// TIA Portal V15.1 export
// export: Created 2020-12-23T11:47:33.918068Z, ExportSetting WithDefaults, WithReadOnly, DisplayName Totally Integrated Automation Portal, DisplayVersion V15.1 Update 3, DisplayName TIA Portal Openness, DisplayVersion V15.1, DisplayName STEP 7 Professional, DisplayVersion V15.1 Update 3, DisplayName WinCC Advanced, DisplayVersion V15.1 Update 3
VAR_GLOBAL   // PLC tag table "io_import"
   "VSEN TBL TABLE LH HP UP" AT I60.0 : Bool;   // #nc - VSEN TBL TABLE LH HP UP
   "VSEN TBL TABLE LH WP DOWN" AT I61.0 : Bool;   // #nc - VSEN TBL TABLE LH WP DOWN
   "VALVE TBL TABLE LH HP UP" AT Q60.6 : Bool;   // [1] VALVE TBL TABLE LH HP UP
   "VALVE TBL TABLE LH WP DOWN" AT Q61.6 : Bool;   // [1] VALVE TBL TABLE LH WP DOWN
   "VSEN TBL TABLE RH HP UP" AT I60.1 : Bool;   // #nc - VSEN TBL TABLE RH HP UP
   "VSEN TBL TABLE RH WP DOWN" AT I61.1 : Bool;   // #nc - VSEN TBL TABLE RH WP DOWN
   "VALVE TBL TABLE RH HP UP" AT Q60.7 : Bool;   // [2] VALVE TBL TABLE RH HP UP
   "VALVE TBL TABLE RH WP DOWN" AT Q61.7 : Bool;   // [2] VALVE TBL TABLE RH WP DOWN
   "VSEN TBL SECTION1 HP UP" AT I20.3 : Bool;   // #nc - VSEN TBL SECTION1 HP UP
   "VSEN TBL SECTION1 WP DOWN" AT I21.3 : Bool;   // #nc - VSEN TBL SECTION1 WP DOWN
   "VALVE TBL SECTION1 HP UP" AT Q40.0 : Bool;   // [3] VALVE TBL SECTION1 HP UP
   "VALVE TBL SECTION1 WP DOWN" AT Q41.0 : Bool;   // [3] VALVE TBL SECTION1 WP DOWN
   "VSEN TBL SECTION2 HP UP" AT I30.3 : Bool;   // #nc - VSEN TBL SECTION2 HP UP
   "VSEN TBL SECTION2 WP DOWN" AT I31.3 : Bool;   // #nc - VSEN TBL SECTION2 WP DOWN
   "VALVE TBL SECTION2 HP UP" AT Q40.1 : Bool;   // [4] VALVE TBL SECTION2 HP UP
   "VALVE TBL SECTION2 WP DOWN" AT Q41.1 : Bool;   // [4] VALVE TBL SECTION2 WP DOWN
   "VSEN TBL SECTION4 LH HP UP" AT I20.4 : Bool;   // #nc - VSEN TBL SECTION4 LH HP UP
   "VSEN TBL SECTION4 LH WP DOWN" AT I21.4 : Bool;   // #nc - VSEN TBL SECTION4 LH WP DOWN
   "VALVE TBL SECTION4 LH HP UP" AT Q40.2 : Bool;   // [5] VALVE TBL SECTION4 LH HP UP
   "VALVE TBL SECTION4 LH WP DOWN" AT Q41.2 : Bool;   // [5] VALVE TBL SECTION4 LH WP DOWN
   "VSEN TBL SECTION4 RH HP UP" AT I30.4 : Bool;   // #nc - VSEN TBL SECTION4 RH HP UP
   "VSEN TBL SECTION4 RH WP DOWN" AT I31.4 : Bool;   // #nc - VSEN TBL SECTION4 RH WP DOWN
   "VALVE TBL SECTION4 RH HP UP" AT Q40.3 : Bool;   // [6] VALVE TBL SECTION4 RH HP UP
   "VALVE TBL SECTION4 RH WP DOWN" AT Q41.3 : Bool;   // [6] VALVE TBL SECTION4 RH WP DOWN
   "VSEN TBL SECTION5 LH HP UP" AT I20.5 : Bool;   // #nc - VSEN TBL SECTION5 LH HP UP
   "VSEN TBL SECTION5 LH WP DOWN" AT I21.5 : Bool;   // #nc - VSEN TBL SECTION5 LH WP DOWN
   "VALVE TBL SECTION5 LH HP UP" AT Q40.4 : Bool;   // [7] VALVE TBL SECTION5 LH HP UP
   "VALVE TBL SECTION5 LH WP DOWN" AT Q41.4 : Bool;   // [7] VALVE TBL SECTION5 LH WP DOWN
   "VSEN TBL SECTION5 RH HP UP" AT I30.5 : Bool;   // #nc - VSEN TBL SECTION5 RH HP UP
   "VSEN TBL SECTION5 RH WP DOWN" AT I31.5 : Bool;   // #nc - VSEN TBL SECTION5 RH WP DOWN
   "VALVE TBL SECTION5 RH HP UP" AT Q40.5 : Bool;   // [8] VALVE TBL SECTION5 RH HP UP
   "VALVE TBL SECTION5 RH WP DOWN" AT Q41.5 : Bool;   // [8] VALVE TBL SECTION5 RH WP DOWN
   "VSEN TBL POSITIONING LH HP UP" AT I20.6 : Bool;   // #nc - VSEN TBL POSITIONING LH HP UP
   "VSEN TBL POSITIONING LH WP DOWN" AT I21.6 : Bool;   // #nc - VSEN TBL POSITIONING LH WP DOWN
   "VALVE TBL POSITIONING LH HP UP" AT Q40.6 : Bool;   // [9] VALVE TBL POSITIONING LH HP UP
   "VALVE TBL POSITIONING LH WP DOWN" AT Q41.6 : Bool;   // [9] VALVE TBL POSITIONING LH WP DOWN
   "VSEN TBL POSITIONING RH HP UP" AT I30.6 : Bool;   // #nc - VSEN TBL POSITIONING RH HP UP
   "VSEN TBL POSITIONING RH WP DOWN" AT I31.5 : Bool;   // #nc - VSEN TBL POSITIONING RH WP DOWN
   "VALVE TBL POSITIONING RH HP UP" AT Q40.7 : Bool;   // [10] VALVE TBL POSITIONING RH HP UP
   "VALVE TBL POSITIONING RH WP DOWN" AT Q41.7 : Bool;   // [10] VALVE TBL POSITIONING RH WP DOWN
   "VSEN TBL PIN LH HP DOWN" AT I20.1 : Bool;   // #nc - VSEN TBL PIN LH HP DOWN
   "VSEN TBL PIN LH WP UP" AT I21.1 : Bool;   // #nc - VSEN TBL PIN LH WP UP
   "VALVE TBL PIN LH HP DOWN" AT Q1000.0 : Bool;   // [11] VALVE TBL PIN LH HP DOWN
   "VALVE TBL PIN LH WP UP" AT Q50.5 : Bool;   // [11] VALVE TBL PIN LH WP UP
   "VSEN TBL PIN RH HP DOWN" AT I30.1 : Bool;   // #nc - VSEN TBL PIN RH HP DOWN
   "VSEN TBL PIN RH WP UP" AT I31.1 : Bool;   // #nc - VSEN TBL PIN RH WP UP
   "VALVE TBL PIN RH HP DOWN" AT Q1000.0 : Bool;   // [12] VALVE TBL PIN RH HP DOWN
   "VALVE TBL PIN RH WP UP" AT Q51.5 : Bool;   // [12] VALVE TBL PIN RH WP UP
   "VSEN TBL SCREW GRIPPER HP OPEN" AT I20.2 : Bool;   // #nc - VSEN TBL SCREW GRIPPER HP OPEN
   "VSEN TBL SCREW GRIPPER WP CLOSE" AT I21.2 : Bool;   // #nc - VSEN TBL SCREW GRIPPER WP CLOSE
   "VALVE TBL SCREW GRIPPER HP OPEN" AT Q1000.0 : Bool;   // [13] VALVE TBL SCREW GRIPPER HP OPEN
   "VALVE TBL SCREW GRIPPER WP CLOSE" AT Q50.4 : Bool;   // [13] VALVE TBL SCREW GRIPPER WP CLOSE
   "VSEN TBL WRAP GRIPPER HP OPEN" AT I20.7 : Bool;   // #nc - VSEN TBL WRAP GRIPPER HP OPEN
   "VSEN TBL WRAP GRIPPER WP CLOSE" AT I21.7 : Bool;   // #nc - VSEN TBL WRAP GRIPPER WP CLOSE
   "VALVE TBL WRAP GRIPPER HP OPEN" AT Q1000.0 : Bool;   // [14] VALVE TBL WRAP GRIPPER HP OPEN
   "VALVE TBL WRAP GRIPPER WP CLOSE" AT Q51.4 : Bool;   // [14] VALVE TBL WRAP GRIPPER WP CLOSE
   "VSEN ST1 POSITIONING HP RIGHT" AT I120.2 : Bool;   // #nc - VSEN ST1 POSITIONING HP RIGHT
   "VSEN ST1 POSITIONING WP LEFT" AT I121.2 : Bool;   // #nc - VSEN ST1 POSITIONING WP LEFT
   "VALVE ST1 POSITIONING HP RIGHT" AT Q120.6 : Bool;   // [15] VALVE ST1 POSITIONING HP RIGHT
   "VALVE ST1 POSITIONING WP LEFT" AT Q121.6 : Bool;   // [15] VALVE ST1 POSITIONING WP LEFT
   "VSEN ST1 SWORD HP OPEN" AT I120.3 : Bool;   // #nc - VSEN ST1 SWORD HP OPEN
   "VSEN ST1 SWORD WP CLOSE" AT I121.3 : Bool;   // #nc - VSEN ST1 SWORD WP CLOSE
   "VALVE ST1 SWORD HP OPEN" AT Q120.7 : Bool;   // [16] VALVE ST1 SWORD HP OPEN
   "VALVE ST1 SWORD WP CLOSE" AT Q121.7 : Bool;   // [16] VALVE ST1 SWORD WP CLOSE
   "VSEN ST2 POSITIONING HP BACK" AT I120.0 : Bool;   // #nc - VSEN ST2 POSITIONING HP BACK
   "VSEN ST2 POSITIONING WP FRONT" AT I121.0 : Bool;   // #nc - VSEN ST2 POSITIONING WP FRONT
   "VALVE ST2 POSITIONING HP BACK" AT Q120.4 : Bool;   // [17] VALVE ST2 POSITIONING HP BACK
   "VALVE ST2 POSITIONING WP FRONT" AT Q121.4 : Bool;   // [17] VALVE ST2 POSITIONING WP FRONT
   "VSEN ST2 SWORD HP UP" AT I120.1 : Bool;   // #nc - VSEN ST2 SWORD HP UP
   "VSEN ST2 SWORD WP DOWN" AT I121.1 : Bool;   // #nc - VSEN ST2 SWORD WP DOWN
   "VALVE ST2 SWORD HP UP" AT Q120.5 : Bool;   // [18] VALVE ST2 SWORD HP UP
   "VALVE ST2 SWORD WP DOWN" AT Q1000.0 : Bool;   // [18] VALVE ST2 SWORD WP DOWN
   "VSEN ST3 POSITIONING HP BACK" AT I140.0 : Bool;   // #nc - VSEN ST3 POSITIONING HP BACK
   "VSEN ST3 POSITIONING WP FRONT" AT 1I41.0 : Bool;   // #nc - VSEN ST3 POSITIONING WP FRONT
   "VALVE ST3 POSITIONING HP BACK" AT Q140.6 : Bool;   // [19] VALVE ST3 POSITIONING HP BACK
   "VALVE ST3 POSITIONING WP FRONT" AT Q141.6 : Bool;   // [19] VALVE ST3 POSITIONING WP FRONT
   "VSEN ST3 SWORD A SQUEEZING HP OPEN" AT I1000.0 : Bool;   // #nc - VSEN ST3 SWORD A SQUEEZING HP OPEN
   "VSEN ST3 SWORD A SQUEEZING WP CLOSE" AT I130.1 : Bool;   // #nc - VSEN ST3 SWORD A SQUEEZING WP CLOSE
   "VALVE ST3 SWORD A SQUEEZING HP OPEN" AT Q1000.0 : Bool;   // [20] VALVE ST3 SWORD A SQUEEZING HP OPEN
   "VALVE ST3 SWORD A SQUEEZING WP CLOSE" AT Q131.4 : Bool;   // [20] VALVE ST3 SWORD A SQUEEZING WP CLOSE
   "VSEN ST3 SWORD A SPREADING HP OPEN" AT I1000.0 : Bool;   // #nc - VSEN ST3 SWORD A SPREADING HP OPEN
   "VSEN ST3 SWORD A SPREADING WP CLOSE" AT I130.0 : Bool;   // #nc - VSEN ST3 SWORD A SPREADING WP CLOSE
   "VALVE ST3 SWORD A SPREADING HP OPEN" AT Q1000.0 : Bool;   // [21] VALVE ST3 SWORD A SPREADING HP OPEN
   "VALVE ST3 SWORD A SPREADING WP CLOSE" AT Q130.5 : Bool;   // [21] VALVE ST3 SWORD A SPREADING WP CLOSE
   "VSEN ST3 SWORD A OPENING HP OPEN" AT I1000.0 : Bool;   // #nc - VSEN ST3 SWORD A OPENING HP OPEN
   "VSEN ST3 SWORD A OPENING WP CLOSE" AT I131.0 : Bool;   // #nc - VSEN ST3 SWORD A OPENING WP CLOSE
   "VALVE ST3 SWORD A OPENING HP OPEN" AT Q1000.0 : Bool;   // [22] VALVE ST3 SWORD A OPENING HP OPEN
   "VALVE ST3 SWORD A OPENING WP CLOSE" AT Q130.4 : Bool;   // [22] VALVE ST3 SWORD A OPENING WP CLOSE
   "VSEN ST3 SWORD B SQUEEZING HP OPEN" AT I1000.0 : Bool;   // #nc - VSEN ST3 SWORD B SQUEEZING HP OPEN
   "VSEN ST3 SWORD B SQUEEZING WP CLOSE" AT I131.2 : Bool;   // #nc - VSEN ST3 SWORD B SQUEEZING WP CLOSE
   "VALVE ST3 SWORD B SQUEEZING HP OPEN" AT Q1000.0 : Bool;   // [23] VALVE ST3 SWORD B SQUEEZING HP OPEN
   "VALVE ST3 SWORD B SQUEEZING WP CLOSE" AT Q131.6 : Bool;   // [23] VALVE ST3 SWORD B SQUEEZING WP CLOSE
   "VSEN ST3 SWORD B SPREADING HP OPEN" AT I1000.0 : Bool;   // #nc - VSEN ST3 SWORD B SPREADING HP OPEN
   "VSEN ST3 SWORD B SPREADING WP CLOSE" AT I131.1 : Bool;   // #nc - VSEN ST3 SWORD B SPREADING WP CLOSE
   "VALVE ST3 SWORD B SPREADING HP OPEN" AT Q1000.0 : Bool;   // [24] VALVE ST3 SWORD B SPREADING HP OPEN
   "VALVE ST3 SWORD B SPREADING WP CLOSE" AT Q130.7 : Bool;   // [24] VALVE ST3 SWORD B SPREADING WP CLOSE
   "VSEN ST3 SWORD B OPENING HP OPEN" AT I1000.0 : Bool;   // #nc - VSEN ST3 SWORD B OPENING HP OPEN
   "VSEN ST3 SWORD B OPENING WP CLOSE" AT I130.2 : Bool;   // #nc - VSEN ST3 SWORD B OPENING WP CLOSE
   "VALVE ST3 SWORD B OPENING HP OPEN" AT Q1000.0 : Bool;   // [25] VALVE ST3 SWORD B OPENING HP OPEN
   "VALVE ST3 SWORD B OPENING WP CLOSE" AT Q130.6 : Bool;   // [25] VALVE ST3 SWORD B OPENING WP CLOSE
   "VSEN ST6 CONNECTOR1 HP UP" AT I150.4 : Bool;   // #nc - VSEN ST6 CONNECTOR1 HP UP
   "VSEN ST6 CONNECTOR1 WP DOWN" AT I151.4 : Bool;   // #nc - VSEN ST6 CONNECTOR1 WP DOWN
   "VALVE ST6 CONNECTOR1 HP UP" AT Q160.4 : Bool;   // [26] VALVE ST6 CONNECTOR1 HP UP
   "VALVE ST6 CONNECTOR1 WP DOWN" AT Q161.4 : Bool;   // [26] VALVE ST6 CONNECTOR1 WP DOWN
   "VSEN ST6 CONNECTOR2 HP UP" AT I150.5 : Bool;   // #nc - VSEN ST6 CONNECTOR2 HP UP
   "VSEN ST6 CONNECTOR2 WP DOWN" AT I151.5 : Bool;   // #nc - VSEN ST6 CONNECTOR2 WP DOWN
   "VALVE ST6 CONNECTOR2 HP UP" AT Q160.5 : Bool;   // [27] VALVE ST6 CONNECTOR2 HP UP
   "VALVE ST6 CONNECTOR2 WP DOWN" AT Q161.5 : Bool;   // [27] VALVE ST6 CONNECTOR2 WP DOWN
   "VSEN ST6 HOLDFAST LH1 HP UP" AT I150.0 : Bool;   // #nc - VSEN ST6 HOLDFAST LH1 HP UP
   "VSEN ST6 HOLDFAST LH1 WP DOWN" AT I151.0 : Bool;   // #nc - VSEN ST6 HOLDFAST LH1 WP DOWN
   "VALVE ST6 HOLDFAST LH1 HP UP" AT Q160.0 : Bool;   // [28] VALVE ST6 HOLDFAST LH1 HP UP
   "VALVE ST6 HOLDFAST LH1 WP DOWN" AT Q161.0 : Bool;   // [28] VALVE ST6 HOLDFAST LH1 WP DOWN
   "VSEN ST6 HOLDFAST LH2 HP UP" AT I150.1 : Bool;   // #nc - VSEN ST6 HOLDFAST LH2 HP UP
   "VSEN ST6 HOLDFAST LH2 WP DOWN" AT I151.1 : Bool;   // #nc - VSEN ST6 HOLDFAST LH2 WP DOWN
   "VALVE ST6 HOLDFAST LH2 HP UP" AT Q160.1 : Bool;   // [29] VALVE ST6 HOLDFAST LH2 HP UP
   "VALVE ST6 HOLDFAST LH2 WP DOWN" AT Q161.1 : Bool;   // [29] VALVE ST6 HOLDFAST LH2 WP DOWN
   "VSEN ST6 HOLDFAST RH1 HP UP" AT I150.2 : Bool;   // #nc - VSEN ST6 HOLDFAST RH1 HP UP
   "VSEN ST6 HOLDFAST RH1 WP DOWN" AT I151.2 : Bool;   // #nc - VSEN ST6 HOLDFAST RH1 WP DOWN
   "VALVE ST6 HOLDFAST RH1 HP UP" AT Q160.2 : Bool;   // [30] VALVE ST6 HOLDFAST RH1 HP UP
   "VALVE ST6 HOLDFAST RH1 WP DOWN" AT Q161.2 : Bool;   // [30] VALVE ST6 HOLDFAST RH1 WP DOWN
   "VSEN ST6 HOLDFAST RH2 HP UP" AT I150.3 : Bool;   // #nc - VSEN ST6 HOLDFAST RH2 HP UP
   "VSEN ST6 HOLDFAST RH2 WP DOWN" AT I151.3 : Bool;   // #nc - VSEN ST6 HOLDFAST RH2 WP DOWN
   "VALVE ST6 HOLDFAST RH2 HP UP" AT Q160.3 : Bool;   // [31] VALVE ST6 HOLDFAST RH2 HP UP
   "VALVE ST6 HOLDFAST RH2 WP DOWN" AT Q161.3 : Bool;   // [31] VALVE ST6 HOLDFAST RH2 WP DOWN
   "VSEN ST6 ROTATION LH HP LEFT" AT I1000.0 : Bool;   // #nc - VSEN ST6 ROTATION LH HP LEFT
   "VSEN ST6 ROTATION LH WP RIGHT" AT I150.6 : Bool;   // #nc - VSEN ST6 ROTATION LH WP RIGHT
   "VALVE ST6 ROTATION LH HP LEFT" AT Q1000.0 : Bool;   // [32] VALVE ST6 ROTATION LH HP LEFT
   "VALVE ST6 ROTATION LH WP RIGHT" AT Q160.6 : Bool;   // [32] VALVE ST6 ROTATION LH WP RIGHT
   "VSEN ST6 ROTATION RH HP RIGHT" AT I1000.0 : Bool;   // #nc - VSEN ST6 ROTATION RH HP RIGHT
   "VSEN ST6 ROTATION RH WP LEFT" AT I151.6 : Bool;   // #nc - VSEN ST6 ROTATION RH WP LEFT
   "VALVE ST6 ROTATION RH HP RIGHT" AT Q1000.0 : Bool;   // [33] VALVE ST6 ROTATION RH HP RIGHT
   "VALVE ST6 ROTATION RH WP LEFT" AT Q161.6 : Bool;   // [33] VALVE ST6 ROTATION RH WP LEFT
END_VAR
